FUNCTION_BLOCK Flasher
VAR_INPUT
	Flash_Frequency : TIME := TIME#10ms;
END_VAR
VAR_OUTPUT
END_VAR
VAR_IN_OUT
	Flasher : INT := 0;
END_VAR
VAR
	// Timer for Flash Function
	Flash_Timer: TON;
END_VAR
VAR // added by the converter: edge detectors and wires of the graphical bodies
    _w1 : BOOL;
END_VAR

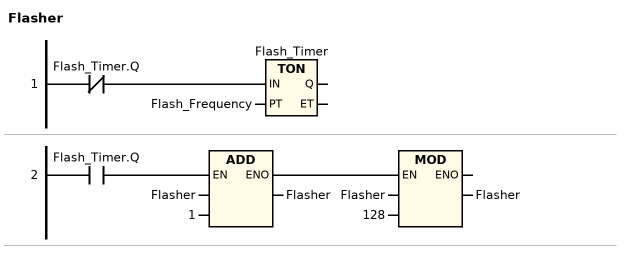
// NETWORK 1
Flash_Timer(IN := NOT Flash_Timer.Q, PT := Flash_Frequency); // TON

// NETWORK 2
_w1 := Flash_Timer.Q;
IF _w1 THEN Flasher := Flasher + 1; END_IF
IF _w1 THEN Flasher := Flasher MOD 128; END_IF

END_FUNCTION_BLOCK

(* stored: Version 1.1.0.1, ProductVersion 3.1.4024.9
   POU Flasher: Id {f5aebd01-51c2-4ff6-8359-ab463684741f}, SpecialFunc None *)
